SUBAPPLICATION NVS_IN_AND_STORE_AR2 (* NVS Laden und Speichern von AR2-Daten mit zusaetzlichem VALUEO (AR, plain) fuer einen weiteren Consumer - da NVS_AR2 keinen eigenen Ausgangs-Plug hat, wird AR_TO_AR2.AR_OUT gesplittet (Q_NumericValue_PHYSA + VALUEO) *)
  (* Standard: 61499-2; Description: Copyright (c) 2026 Meisterschulen am Ostbahnhof This program and the accompanying materials are made available under the terms of the Eclipse Public License 2.0 which is available at https://www.eclipse.org/legal/epl-2.0/ SPDX-License-Identifier: EPL-2.0 *)
  (* Version 1.0, 2026-08-31, Franz Höpfinger, Meisterschulen am Ostbahnhof, AR2 adapter variant of NVS_IN_AND_STORE_AR - NumericValue_PHYSA + AR_TO_AR2 + NVS_AR2 (Speicherung via AR2 Socket), AR_TO_AR2.AR_OUT gesplittet auf Q_NumericValue_PHYSA (VT-Anzeige) und VALUEO (weiterer Consumer) *)
  PACKAGE MyLib::sys;
  IMPORT isobus::UT::Q::const::IDs::ID_NULL;
  IMPORT logiBUS::utils::conversion::phys::NumericObjectPool_S;
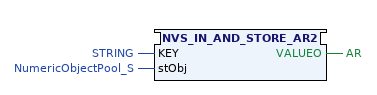
  VAR_INPUT
    KEY : STRING; (* Key name. *)
    stObj : logiBUS::utils::conversion::phys::NumericObjectPool_S := (u16ObjId := ID_NULL, r32Scale := 1.0, i32Offset := 0, u8Decimals := 0);
  END_VAR
  PLUGS
    VALUEO : adapter::types::unidirectional::AR;
  END_PLUGS
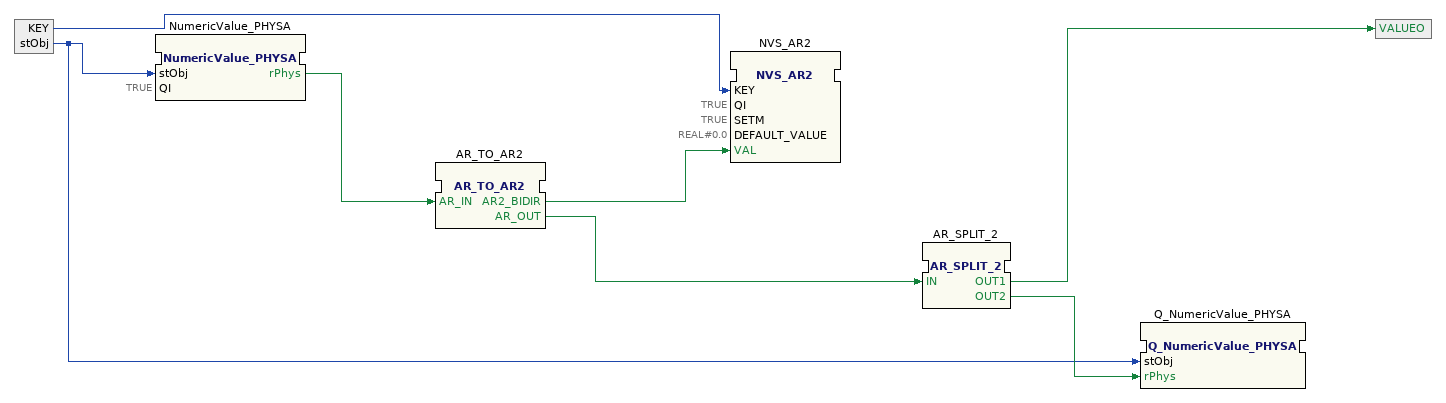
  (* SETM=TRUE - der Boot-Wert laedt so oder so automatisch (INIT -> INITO -> GET -> GETO, unabhaengig von SETM). SETM=TRUE sorgt dafuer, dass auch eine LIVE-Aenderung waehrend des laufenden Betriebs sofort bestaetigt/zurueckgemeldet wird - wichtig, falls der frische Wert noch im selben Lauf weiterverwendet werden soll (z.B. hier ueber VALUEO). *)
  FBS
    NumericValue_PHYSA : isobus::UT::io::NumericValue::NumericValue_PHYSA(QI := TRUE);
    AR_TO_AR2 : adapter::conversion::bidirectional::AR_TO_AR2;
    NVS_AR2 : logiBUS::storage::esp32_nvs::NVS_AR2(QI := TRUE, SETM := TRUE, DEFAULT_VALUE := REAL#0.0);
    AR_SPLIT_2 : adapter::events::unidirectional::AR_SPLIT_2;
    Q_NumericValue_PHYSA : isobus::UT::Q::Q_NumericValue_PHYSA;
  END_FBS
  DATA_CONNECTIONS
    stObj TO Q_NumericValue_PHYSA.stObj;
    KEY TO NVS_AR2.KEY;
    stObj TO NumericValue_PHYSA.stObj;
  END_CONNECTIONS
  ADAPTER_CONNECTIONS
    NumericValue_PHYSA.rPhys TO AR_TO_AR2.AR_IN;
    AR_TO_AR2.AR2_BIDIR TO NVS_AR2.VAL;
    AR_TO_AR2.AR_OUT TO AR_SPLIT_2.IN;
    AR_SPLIT_2.OUT1 TO VALUEO;
    AR_SPLIT_2.OUT2 TO Q_NumericValue_PHYSA.rPhys;
  END_CONNECTIONS
END_SUBAPPLICATION
